FUNCTION_BLOCK FB_SafetyCompositionCustomized
VAR_INPUT
	///true if initializing is active
	_InitSafety: BOOL;
END_VAR


IF(_InitSafety) Then
	//Add project specific safety code that shall execute during PLC init/reinit. 
	;
ELSE
	//Add project specific safety code here. 
	//renamed from Com_Error to FB_SafetyCompositionCustomized
	;
END_IF

END_FUNCTION_BLOCK

(* stored: Version 1.1.0.1, ProductVersion 3.1.4024.9
   POU FB_SafetyCompositionCustomized: Id {065010de-5397-4e15-b987-4489b2f1ef56}, SpecialFunc None *)
